FUNCTION_BLOCK FB_HMI_VOTER EXTENDS FB_HMI_COMPONENT
VAR_INPUT
END_VAR
VAR_OUTPUT
END_VAR
VAR_IN_OUT
    fbInstance : FB_METIS_VOTER;
END_VAR
VAR
END_VAR

fbHealthStatus(
    bIsEnabled := fbInstance.stat.bEnabled,
    bIsGood := fbInstance.stat.bValid);
                     
fbBusyStatus(
    bIsEnabled := FALSE,
    bIsBusy := FALSE);

M_UpdateStatusColor();

END_FUNCTION_BLOCK

(* stored: Version 1.1.0.1, ProductVersion 3.1.4024.14
   POU FB_HMI_VOTER: Id {f7de15b8-a306-4cd7-a559-6c87017aadef}, SpecialFunc None *)
